Staubli VAL3: JointSpace.dtx

public jointRx JointPos
public num JointVel[6]
public num JointAccel[6]
public num JointForce[6]
